ABB RAPID module: MainModule.mod

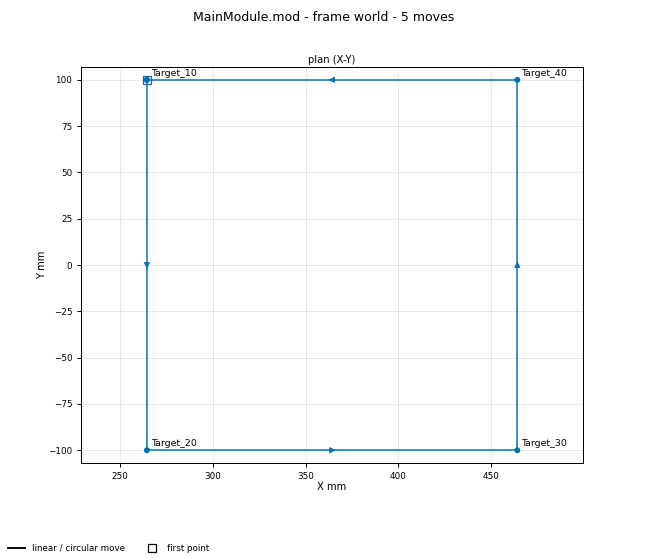
[picture p0: tool path of MainModule.mod in frame world, 5 of 5 moves have a stored position in this frame; points joined in program order, loops and branches not executed]
MODULE MainModule
        CONST robtarget Target_10:=[[264.350012476,100.000011179,593.999948019],[0.500000001,0.000000007,0.866025403,0],[0,-1,0,0],[9E+09,9E+09,9E+09,9E+09,9E+09,9E+09]];
    CONST robtarget Target_20:=[[264.350012476,-100.000011179,593.999948019],[0.500000001,-0.000000007,0.866025403,0],[-1,0,-1,0],[9E+09,9E+09,9E+09,9E+09,9E+09,9E+09]];
    CONST robtarget Target_30:=[[464.350000726,-100.00000079,593.999945781],[0.500000003,-0.000000003,0.866025402,0.000000005],[-1,0,-1,0],[9E+09,9E+09,9E+09,9E+09,9E+09,9E+09]];
    CONST robtarget Target_40:=[[464.350000726,100.00000079,593.999945781],[0.500000003,0.000000003,0.866025402,-0.000000005],[0,-1,0,0],[9E+09,9E+09,9E+09,9E+09,9E+09,9E+09]];
    CONST robtarget Target_50:=[[264.350012476,100.000011179,593.999948019],[0.500000001,0.000000007,0.866025403,0],[0,-1,0,0],[9E+09,9E+09,9E+09,9E+09,9E+09,9E+09]];
!***********************************************************
    !
    ! Module:  MainModule
    !
    ! Description:
    !   <Insert description here>
    !
    ! Author: niels
    !
    ! Version: 1.0
    !
    !***********************************************************


    !***********************************************************
    !
    ! Procedure main
    !
    !   This is the entry point of your program
    !
    !***********************************************************
    PROC main()
        Path_10;
    ENDPROC
    PROC Path_10()
        MoveJ Target_10,v400,z50,tool0\WObj:=wobj0;
        MoveL Target_20,v100,z50,tool0\WObj:=wobj0;
        MoveL Target_30,v100,z50,tool0\WObj:=wobj0;
        MoveL Target_40,v100,z50,tool0\WObj:=wobj0;
        MoveL Target_50,v100,z50,tool0\WObj:=wobj0;
    ENDPROC
ENDMODULE
